FUNCTION_BLOCK FB_CoE_Write
VAR_INPUT
	// Link this to your terminal's drive reference variables under InfoData.
	stPlcDriveRef : ST_PlcDriveRef;
END_VAR
VAR_OUTPUT
END_VAR
VAR
	// Write Error
	bWriteError : BOOL;
	// Data successfully sent
	bDataSent : BOOL := FALSE;
	
	fbCoeWrite: FB_CoEWrite_ByDriveRef;
	
	stDriveRef: ST_DriveRef;
	
	nState : BYTE := 0;   //State Machine
END_VAR

stDriveRef.sNetId := F_CreateAmsNetId(stPlcDriveRef.aNetId);
stDriveRef.nSlaveAddr := stPlcDriveRef.nSlaveAddr;
stDriveRef.nDriveNo := stPlcDriveRef.nDriveNo;
stDriveRef.nDriveType := stPlcDriveRef.nDriveType;

CASE nState OF
	0: //Idle state
		HandleIdle();
	1: //Writing data
		HandleWritingData();
	100: //Handle Error
		HandleError();
END_CASE

ACTION HandleError:
// wait for reset ccmmand
bDataSent := FALSE;
END_ACTION

ACTION HandleIdle:
fbCoeWrite(bExecute := FALSE);
// Reset DataSent bit
bDataSent := FALSE;
END_ACTION

ACTION HandleWritingData:
fbCoeWrite(bExecute := TRUE);       // Execute CoE write until done
IF fbCoeWrite.bError THEN
	nState := 100;     // Error case
	bWriteError := TRUE;
ELSE
	IF NOT fbCoeWrite.bBusy THEN
		nState := 0;    // Done
		bDataSent := TRUE;
	END_IF
END_IF
END_ACTION

METHOD InErrorState : BOOL
VAR_INPUT
END_VAR
IF nState = 100 THEN
	InErrorState := TRUE;
ELSE
	InErrorState := FALSE;
END_IF
END_METHOD

METHOD IsBusy : BOOL
VAR_INPUT
END_VAR
IF nState <> 0 THEN
	IsBusy := TRUE;
ELSE
	IsBusy := FALSE;
END_IF
END_METHOD

PROPERTY IsDataSent : BOOL
GET
IsDataSent := bDataSent;
END_GET
END_PROPERTY

METHOD ResetError
VAR_INPUT
END_VAR
IF nState <> 100 THEN
	RETURN;
END_IF

// Reset write error
bWriteError := FALSE;
// Go to Idle state
nState := 0;
END_METHOD

METHOD WriteData
VAR_INPUT
	//stCoeParameter : ST_CoeParameter;
	nIndex: WORD;
	// Hexadecimal subindex of CoE, e.g. the 12 in 8010:12
	nSubIndex: BYTE;
	// Pointer to a value to fill with the result of the read, e.g. ADR(MyValue)
	pSrcBuf: PVOID;
	// Data size of pSrcBuf, e.g. SIZEOF(MyValue)
	cbBufLen: UDINT;
END_VAR
IF nState <> 0 THEN
	RETURN;
END_IF

fbCoeWrite(
	stDriveRef := stDriveRef,
	nIndex := nIndex,
	nSubIndex := nSubIndex,
	pSrcBuf := pSrcBuf,
	cbBufLen := cbBufLen,
	tTimeout := T#1S,
);

// Go to Writing Data state
nState := 1;
END_METHOD

END_FUNCTION_BLOCK

(* stored: Version 1.1.0.1, ProductVersion 3.1.4022.18
   POU FB_CoE_Write: Id {dd0856f6-a4c1-470a-beca-fb09638dc24b}, SpecialFunc None
   Action HandleError: Id {98f20886-2ef9-4d63-917f-95e80c4ac5cf}
   Action HandleIdle: Id {20ca62bf-ad0a-4177-a59e-8311ad0fb51b}
   Action HandleWritingData: Id {f1cec576-6950-4b61-b35d-05dc9178ea43}
   Method InErrorState: Id {9116d509-8999-416b-adbd-60527b13a43a}
   Method IsBusy: Id {508a4fdc-b906-4ba8-8612-c854593be8cf}
   Property IsDataSent: Id {8a6f48ef-d77e-4d1b-bd8d-3fcf65210096}
   Get Get: Id {0f6d758f-97ac-411f-95f2-181644180e78}
   Method ResetError: Id {a0677d16-b2a2-49d4-8dfc-d9f483828e92}
   Method WriteData: Id {2540e6f5-2c02-45e8-b017-e09b99229358} *)
